# EPICS IOC start-up script: iocsh/io.iocsh
# ### io.iocsh ###

#- ###################################################
#- PREFIX           - IOC Prefix
#- MONO             - Monochrometer positioner field
#- VSC              - Associated scan record
#- OPTICS           - Location of optics module
#- ###################################################

#- Io calculation
dbLoadRecords("$(OPTICS)/opticsApp/Db/Io.db","P=$(PREFIX)Io:")
doAfterIocInit("seq &Io, 'P=$(PREFIX)Io:,MONO=$(MONO),VSC=$(VSC)'")
